			stRotationOptions.additionalTurns := 0;
			stRotationOptions.direction		  := Tc3_Mc3PlanarMotion.MC_Direction.mcDirectionNonModulo;

			IF NOT ipMoverApplication[nMoverIndex].std.P_MoveC.Busy THEN
					
				ipMoverApplication[nMoverIndex].std.MoveC( strInfo,
														   fRotationAngle,
														   fRotationVelocity,
														   fRotationAcceleration,
														   fRotationAcceleration,
														   fRotationJerk,
														   stRotationOptions );
														   
				nStateProcess := nStateProcess +1;
			END_IF										   

	211:	// Checking move command return
			IF ipMoverApplication[nMoverIndex].std.P_MoveC.Done THEN
				nStateProcess := nStateProcess +9;
			ELSIF ipMoverApplication[nMoverIndex].std.P_MoveC.Error THEN
				   nErrorID := ipMoverApplication[nMoverIndex].std.P_MoveOnTrack.ErrorID;
				  nObjectID := ipMoverApplication[nMoverIndex].std.P_MoveOnTrack.stInfo.nObjectID;
				nObjectType := ipMoverApplication[nMoverIndex].std.P_MoveOnTrack.stInfo.nObjectType;				
			END_IF			
			
				
	220:	// Process: Rotation-Demo done
			nStateProcess := 300;

		
			
			
	300: 	// Send mover to the next station
			fMoverToTrackPosition   := fSendAwayPosition;	
			nTrackIndex        		:= nStationTrackIndex;		
			fMoverVelocity     		:=    300.0;
			fMoverAcceleration 		:=  1_000.0;
			fMoverJerk         		:= 10_000.0;	
	
			
			stMoveParameters.direction := Tc3_Mc3PlanarMotion.MC_DIRECTION.mcDirectionPositive;	
			stMoveParameters.gap       := 240.0;

			
			// Creating info text with a little history of what happened in the station for debugging purpose		
			strInfo := fbHistoryInfo.CreateStationInfo(nStationIndex, nMoverIndex, nNextStationIndex);	
			
				
			// Move on track command	
			ipMoverApplication[nMoverIndex].std.MoveOnTrack( strInfo,
															 ipTrack[nTrackIndex].std,
															 fMoverToTrackPosition,
															 fMoverVelocity,
															 fMoverAcceleration,
															 fMoverJerk,
															 stMoveParameters.gap,
															 stMoveParameters.direction);
			nStateProcess := nStateProcess +1;
			
		
		
	301: 	// Checking move command return
			IF ipMoverApplication[nMoverIndex].std.P_MoveOnTrack.Active
			OR ipMoverApplication[nMoverIndex].std.P_MoveOnTrack.Done 
			THEN
				nStateProcess := nStateProcess + 9;
				
			ELSIF ipMoverApplication[nMoverIndex].std.P_MoveOnTrack.Error THEN
				   nErrorID := ipMoverApplication[nMoverIndex].std.P_MoveOnTrack.ErrorID;
				  nObjectID := ipMoverApplication[nMoverIndex].std.P_MoveOnTrack.stInfo.nObjectID;
				nObjectType := ipMoverApplication[nMoverIndex].std.P_MoveOnTrack.stInfo.nObjectType;
			END_IF		
		
			
	310: 	// Mover to the list of the next station
			ipStation[nNextStationIndex].P_List_Switch_Input_C.AddMover(P_List_Station.RemoveFirstInList());
			nStateProcess := 500;	
	
		
	500: 	// Done for this cycle
			nStateProcess := 100;

END_CASE
END_METHOD

END_FUNCTION_BLOCK

// ---- 2_Application/Station/FB_Station_03_Process.TcPOU
FUNCTION_BLOCK FB_Station_03_Process EXTENDS FB_StationBase
VAR
	nStationIndex				: UINT;
	nNextStationIndex			: UINT;
	nStationTrackIndex			: UINT;
	
	fStationPosition_X 			: LREAL;
	fStationPosition_Y 			: LREAL;		  
    fSendAwayDistance			: LREAL;	
	fInRangeDistance			: LREAL;	
	fSendAwayPosition			: LREAL;
	
	position					: PositionXYC;

END_VAR

METHOD Clear : BOOL
VAR_INPUT
END_VAR



	CASE nStateClear OF
		
	0:	// Enter
		Clear := FALSE;
		nStateClear := nStateClear +10;
		
	10: // Clearing all Station-Lists 
		IF SUPER^.Clear() THEN
			nStateClear := nStateClear +10;
		END_IF	
	
	20:	// Add aditional Data to be cleared here...
		nStateClear := 100;
		
		
	100: // Done
		      Clear := TRUE;
		nStateClear := 0;

	END_CASE
END_METHOD

METHOD Init : BOOL



VAR_INST
	nTestCounter	: INT;	
END_VAR
nTestCounter := nTestCounter +1;

CASE nStateInit OF

	0:		// Enter 
			bStationInitDone := FALSE;
			   nStateProcess := 0;
			      nStateInit := 10;
				 
			
	10:		// Init Station-Parameters				
				  nStationIndex := 3;				// Each station needs an unique index	
			 nStationTrackIndex := 3;	 			// Track on which the station resides
			  nNextStationIndex := 5;				// Index of the following station 
							  
			 fStationPosition_X := 840.0;			// Position of the station in X/Y coordinates
			 fStationPosition_Y := 360.0;			// Position of the station in X/Y coordinates
			  
			  fSendAwayDistance := 300.0;			// Position on track a mover will be send to after processing 
			  fInRangeDistance  := 300.0;			// Position in front of a station from where a mover will be taken over
			  
			  nStateInit := 11;
				   
				  
	11: // Fail-safe check, just to make sure all variables have been assigned after doing copy&paste from the template
			IF        nStationIndex > 0
			AND  nStationTrackIndex > 0
			AND   nNextStationIndex > 0
			AND  fStationPosition_X > 0
			AND  fStationPosition_Y > 0
			AND   fSendAwayDistance > 0
			THEN   
				nStateInit := 20;
			END_IF
			
				   
	20:		// Calculating positions
	
			// 1. Calculating station position on track
			position.SetValuesXYC(fStationPosition_X, fStationPosition_Y, 0.0);
			fStationPositionOnTrack := ipTrack[nStationTrackIndex].std.GetTrackPositionAt(position);
							
			// 2. Calculating send-away position on track
			fSendAwayPosition := fStationPositionOnTrack + fSendAwayDistance; 
			
			// The send away position must not exceed the lenght of the track!
			IF fSendAwayPosition > ipTrack[nStationTrackIndex].P_TrackLength THEN
				fSendAwayPosition := ipTrack[nStationTrackIndex].P_TrackLength;
			END_IF
			
			// 3. Calculating the station position in X/Y coordinates determined by the track	
            //    This is to make sure the center of the station is always located directly on the track.
			//    This value can differ from the initial fStationPosition_X, fStationPosition_Y in case they were not matching the track
			ipTrack[nStationTrackIndex].std.GetMoverPositionAt(fStationPositionOnTrack, StationPosition);
			
			// Providing the station position to e.g. visualization	
			stStationPosition.bInit            := TRUE;
			stStationPosition.fPositionOnTrack := fStationPositionOnTrack;
			stStationPosition.nTrackId         := nStationTrackIndex;
			stStationPosition.fPosition_X	   := StationPosition.x;
			stStationPosition.fPosition_Y	   := StationPosition.y;

			nStateInit := 30;
			
			
	30:		// Clear Lists
			IF THIS^.Clear() THEN
				nStateInit := 90;	
			END_IF

			
		
	90:		// Creating a little history of what happened in the station for debugging purpose
			fbHistoryInfo.AddEntry('Init');
	
			nStateInit := 100;
			
						
	100:	// Init done
			IF SUPER^.Init() THEN
				bStationInitDone := TRUE;	
				           Init := TRUE;
			END_IF
				
	
END_CASE
END_METHOD

METHOD Process : BOOL

VAR_INST
		
	nMoverIndex				: UINT;
	
	fMoverToTrackPosition	: LREAL;
	nTrackIndex				: UINT;
	fMoverVelocity			: LREAL;
	fMoverAcceleration		: LREAL;
	fMoverJerk				: LREAL;
	
	
	nErrorId					: UDINT;
	nObjectID					: UDINT;
	nObjectType					: UDINT;		
	
	// Process
	Timer01						: TON;
	fRotationAngle				: LREAL;
	fRotationVelocity			: LREAL;	
	fRotationAcceleration		: LREAL;
	fRotationJerk				: LREAL;
	stRotationOptions			: ST_MoveCOptions;
	
	fbRandom					: DRAND;
	fRandom						: LREAL;
	nRandom						: INT;
	
	bMoverGoodToGo				: BOOL;
	
	
	
END_VAR




VAR_INST



//	bToggleSwitch				: BOOL;
//	bStationActive				: BOOL;


//	fPositionOnTrack			: LREAL;
//	nCurrentTrackIndex			: UDINT;
	


//	fInRangePosition			: LREAL;
//	fOutOfRangePosition			: LREAL;
	


	
	
	
//	strInfo						: STRING;
	
					
	

//	ClearTrig					: R_TRIG;
	
//	TrackInfo					: PlanarObjectInfo;
//	nStationTrackID				: UDINT;
//	nMoverOnTrackID				: UDINT;
	

	
//	stMoveOptionsCurve			: ST_MoveCOptions;
//	fVeloTurn           		: LREAL :=   180.0;
//	fAccelTurn    				: LREAL :=  1000.0;
//	fJerkTurn            		: LREAL := 10000.0;	
//	fTurnAngle					: LREAL;	
	

END_VAR


// *** Processing Station ***

CASE nStateProcess OF 

	0:		// Enter
			IF bStationInitDone THEN
				nStateProcess := 100;
			END_IF

	
	100: 	// Waiting for Mover
			IF P_List_Station.P_FirstInList <> 0 THEN
				nMoverIndex := P_List_Station.P_FirstInList.P_Id;
					 nStateProcess := nStateProcess +10;
			END_IF
	
		
	110: 	// Check if Mover is in range
			IF  ipMoverApplication[nMoverIndex].std.P_SetOnTrack.TrackOID = ipTrack[nStationTrackIndex].std.P_OID 
			AND ipMoverApplication[nMoverIndex].std.P_SetOnTrack.SetPos   > fStationPositionOnTrack - fInRangeDistance
			THEN
				nStateProcess := nStateProcess +10;
			END_IF
			
	
	120: 	// Checking process situation
			CASE eProcessMode OF
				
			E_ProcessMode.None:
				;	// Nothing happens -> Process mode needs to be set!
				
			E_ProcessMode.InitRun:
				IF nStationIndex = 1 THEN
					ipMoverApplication[nMoverIndex].P_ProductData.bInitRun := FALSE;
				ELSE
					nStateProcess := 300;
				END_IF				
			
			E_ProcessMode.Production:
				nStateProcess := 200;
		
			END_CASE
		
	
	200: 	// Send mover to Processing-Position
			fMoverToTrackPosition   := fStationPositionOnTrack;
			nTrackIndex        		:= nStationTrackIndex;
			fMoverVelocity     		:=    300.0;
			fMoverAcceleration 		:=  1_000.0;
			fMoverJerk         		:= 10_000.0;	
	
			stMoveParameters.direction := Tc3_Mc3PlanarMotion.MC_DIRECTION.mcDirectionShortestWay;
			stMoveParameters.gap       := 200.0;
		
			
			// Creating info text with a little history of what happened in the station for debugging purpose		
			strInfo := fbHistoryInfo.CreateStationInfo(nStationIndex, nMoverIndex, nNextStationIndex);	


			// Move on track command	
			ipMoverApplication[nMoverIndex].std.MoveOnTrack( strInfo,
															 ipTrack[nTrackIndex].std,
															 fMoverToTrackPosition,
															 fMoverVelocity,
															 fMoverAcceleration,
															 fMoverJerk,
															 stMoveParameters.gap,
															 stMoveParameters.direction);
			nStateProcess := nStateProcess +1;
				
			
	201: 	// Checking move command return
			IF ipMoverApplication[nMoverIndex].std.P_MoveOnTrack.Done THEN
				nStateProcess := nStateProcess +9;
			ELSIF ipMoverApplication[nMoverIndex].std.P_MoveOnTrack.Error THEN
				   nErrorID := ipMoverApplication[nMoverIndex].std.P_MoveOnTrack.ErrorID;
				  nObjectID := ipMoverApplication[nMoverIndex].std.P_MoveOnTrack.stInfo.nObjectID;
				nObjectType := ipMoverApplication[nMoverIndex].std.P_MoveOnTrack.stInfo.nObjectType;
			END_IF		

			
	210:	// Process: Showing mover rotation -> Rotating 180°
			IF nRandom = 0 THEN
				fbRandom(seed := 0, Num=>fRandom);
				nRandom := LREAL_TO_INT(10*fRandom);
				nRandom := MAX(2,nRandom);
				IF nRandom > 8 THEN
					nRandom := -4;
				END_IF
			END_IF
			
			
			
			       fRotationAngle :=   90.0 * nRandom;
			    fRotationVelocity :=  360.0;
			fRotationAcceleration := 1800.0;
			        fRotationJerk := 9000.0;

			stRotationOptions.additionalTurns := 0;
			stRotationOptions.direction		  := Tc3_Mc3PlanarMotion.MC_Direction.mcDirectionNonModulo;

			IF NOT ipMoverApplication[nMoverIndex].std.P_MoveC.Busy THEN
					
				ipMoverApplication[nMoverIndex].std.MoveC( strInfo,
														   fRotationAngle,
														   fRotationVelocity,
														   fRotationAcceleration,
														   fRotationAcceleration,
														   fRotationJerk,
														   stRotationOptions );
				
			   	      nRandom := 0;										   
				nStateProcess := nStateProcess +1;
			END_IF										   

	211:	// Checking move command return
			IF ipMoverApplication[nMoverIndex].std.P_MoveC.Done THEN
				nStateProcess := nStateProcess +9;
			ELSIF ipMoverApplication[nMoverIndex].std.P_MoveC.Error THEN
				   nErrorID := ipMoverApplication[nMoverIndex].std.P_MoveOnTrack.ErrorID;
				  nObjectID := ipMoverApplication[nMoverIndex].std.P_MoveOnTrack.stInfo.nObjectID;
				nObjectType := ipMoverApplication[nMoverIndex].std.P_MoveOnTrack.stInfo.nObjectType;				
			END_IF			
			
				
	220:	// Process: Rotation-Demo done
			nStateProcess := 300;

				
	300:	// Check if the next station is ready to receive a mover
			IF eProcessMode = E_ProcessMode.Production THEN
				IF ipStation[nNextStationIndex].P_ProcessClearance = 0 THEN
					ipStation[nNextStationIndex].P_ProcessRequest := nStationIndex;
					nStateProcess := nStateProcess +1;	
				END_IF					
			ELSE
				nStateProcess := nStateProcess +10;
			END_IF
	
	301:	IF ipStation[nNextStationIndex].P_ProcessClearance = nStationIndex THEN
				nStateProcess := nStateProcess +9;	
			ELSIF ipStation[nNextStationIndex].P_ProcessRequest <> nStationIndex THEN
				nStateProcess := nStateProcess -1;
			END_IF
					
		
	310: 	// Send mover to the next station
			fMoverToTrackPosition   := fSendAwayPosition;	
			nTrackIndex        		:= nStationTrackIndex;		
			fMoverVelocity     		:=    300.0;
			fMoverAcceleration 		:=  1_000.0;
			fMoverJerk         		:= 10_000.0;	
	
			
			stMoveParameters.direction := Tc3_Mc3PlanarMotion.MC_DIRECTION.mcDirectionPositive;	
			stMoveParameters.gap       := 240.0;

			
			// Creating info text with a little history of what happened in the station for debugging purpose		
			strInfo := fbHistoryInfo.CreateStationInfo(nStationIndex, nMoverIndex, nNextStationIndex);	
			
				
			// Move on track command	
			ipMoverApplication[nMoverIndex].std.MoveOnTrack( strInfo,
															 ipTrack[nTrackIndex].std,
															 fMoverToTrackPosition,
															 fMoverVelocity,
															 fMoverAcceleration,
															 fMoverJerk,
															 stMoveParameters.gap,
															 stMoveParameters.direction);
			nStateProcess := nStateProcess +1;
			
		
		
	311: 	// Checking move command return
			IF ipMoverApplication[nMoverIndex].std.P_MoveOnTrack.Active
			OR ipMoverApplication[nMoverIndex].std.P_MoveOnTrack.Done 
			THEN
				nStateProcess := nStateProcess + 9;
				
			ELSIF ipMoverApplication[nMoverIndex].std.P_MoveOnTrack.Error THEN
				   nErrorID := ipMoverApplication[nMoverIndex].std.P_MoveOnTrack.ErrorID;
				  nObjectID := ipMoverApplication[nMoverIndex].std.P_MoveOnTrack.stInfo.nObjectID;
				nObjectType := ipMoverApplication[nMoverIndex].std.P_MoveOnTrack.stInfo.nObjectType;
			END_IF		
		
			
	320: 	// Mover to the list of the next station
			ipStation[nNextStationIndex].P_List_Switch_Input_B.AddMover(P_List_Station.RemoveFirstInList());
			nStateProcess := 500;	
	
		
	500: 	// Done for this cycle
			nStateProcess := 100;

END_CASE
END_METHOD

END_FUNCTION_BLOCK

// ---- 2_Application/Station/FB_Station_04_SW_Separate.TcPOU
FUNCTION_BLOCK FB_Station_04_SW_Separate EXTENDS FB_StationBase

VAR
	nStationIndex				: UINT;
	nPreviousStationIndexInputA : UINT;	
	nTrackIndexInputA 			: UINT;		
	nNextStationIndexOutputB 	: UINT;	
	nTrackIndexOutputB 			: UINT;		
	nNextStationIndexOutputC 	: UINT;	
	nTrackIndexOutputC 			: UINT;		
	
	fStationPosition_X 			: LREAL;
	fStationPosition_Y 			: LREAL;
	fInRangeDistance			: LREAL;		  
    fSendAwayDistanceOutputB    : LREAL;
	fSendAwayDistanceOutputC    : LREAL;	
	fSendAwayPositionOutputB	: LREAL;
	fSendAwayPositionOutputC	: LREAL;	

	position					: PositionXYC;

END_VAR

METHOD Clear : BOOL
VAR_INPUT
END_VAR



	CASE nStateClear OF
		
	0:	// Enter
		Clear := FALSE;
		nStateClear := nStateClear +10;
		
	10: // Clearing all Station-Lists 
		IF SUPER^.Clear() THEN
			nStateClear := nStateClear +10;
		END_IF	
	
	20:	// Add aditional Data to be cleared here...
		nStateClear := 100;
		
		
	100: // Done
		      Clear := TRUE;
		nStateClear := 0;

	END_CASE
END_METHOD

METHOD Init : BOOL



VAR_INST
	nTestCounter	: INT;	
END_VAR
nTestCounter := nTestCounter +1;

CASE nStateInit OF

	0:		// Enter 
			bStationInitDone := FALSE;
			   nStateProcess := 0;
			      nStateInit := 10;
				 
			
	10:		// Init Station-Parameters				
					       nStationIndex := 4;		// Each station needs an unique index		
			 nPreviousStationIndexInputA := 1;		// Index of the previous station on input_A		
				       nTrackIndexInputA := 1;		// Track on which the previous station resides	
			    nNextStationIndexOutputB := 3;		// Index of the following station on output_B		
				      nTrackIndexOutputB := 3;		// Track on which the following station resides
			    nNextStationIndexOutputC := 2;		// Index of the following station on output_C	
				      nTrackIndexOutputC := 2;		// Track on which the following station resides	 
			
                    fInRangeDistance := 300.0;		// Position in front of a station from where a mover will be taken over			  
		    fSendAwayDistanceOutputB := 300.0;		// Position on track a mover will be send to after processing 
		    fSendAwayDistanceOutputC := 300.0;		// Position on track a mover will be send to after processing 
		
			  nStateInit := 11;

			   
	11: // Fail-safe check, just to make sure all variables have been assigned after doing copy&paste from the template
			IF              nStationIndex > 0
			AND   nPreviousStationIndexInputA > 0	
			AND         nTrackIndexInputA > 0
			AND  nNextStationIndexOutputB > 0
			AND        nTrackIndexOutputB > 0
			AND  nNextStationIndexOutputC > 0
			AND        nTrackIndexOutputC > 0					
			AND          fInRangeDistance > 0
			AND  fSendAwayDistanceOutputB > 0
			AND  fSendAwayDistanceOutputC > 0
			THEN   
				nStateInit := 20;
			END_IF
			
				   
	20:		// Calculating positions
	
			// 1. Calculating station position on track
			fStationPositionOnTrack := ipTrack[nTrackIndexInputA].P_TrackLength;
							
			// 2. Calculating send-away position on track
			fSendAwayPositionOutputB := fSendAwayDistanceOutputB; 
			fSendAwayPositionOutputC := fSendAwayDistanceOutputC;
			
			// The send away position must not exceed the lenght of the following track!
			fSendAwayPositionOutputB := MIN(fSendAwayPositionOutputB, ipTrack[nTrackIndexOutputB].P_TrackLength);
			fSendAwayPositionOutputC := MIN(fSendAwayPositionOutputC, ipTrack[nTrackIndexOutputC].P_TrackLength);
			
					
			// 3. Calculating the station position in X/Y coordinates determined by the track	
            //    This is to make sure the center of the station is always located directly on the track.
			ipTrack[nTrackIndexInputA].std.GetMoverPositionAt(fStationPositionOnTrack, StationPosition);
			
			// Providing the station position to e.g. visualization	
			stStationPosition.bInit            := TRUE;
			stStationPosition.fPositionOnTrack := fStationPositionOnTrack;
			stStationPosition.nTrackId         := nTrackIndexOutputB;
			stStationPosition.fPosition_X	   := StationPosition.x;
			stStationPosition.fPosition_Y	   := StationPosition.y;

			nStateInit := 30;
			
			
	30:		// Clear Lists
			IF THIS^.Clear() THEN
				nStateInit := 90;	
			END_IF

			
		
	90:		// Creating a little history of what happened in the station for debugging purpose
			fbHistoryInfo.AddEntry('Init');
	
			nStateInit := 100;
			
						
	100:	// Init done
			IF SUPER^.Init() THEN
				bStationInitDone := TRUE;	
				           Init := TRUE;
			END_IF
				
	
END_CASE
END_METHOD

METHOD Process : BOOL

VAR_INST
		
	nMoverIndex				: UINT;
	
	fMoverToTrackPosition	: LREAL;
	nTrackIndex				: UINT;
	fMoverVelocity			: LREAL;
	fMoverAcceleration		: LREAL;
	fMoverJerk				: LREAL;
	
	
	nErrorId				: UDINT;
	nObjectID				: UDINT;
	nObjectType				: UDINT;		
	
	
	// Process
	nDestinationProcess		: UINT;
	nIncommingTrackOID		: UDINT;
	nNextStationIndex		: UINT;		 				
	fSendAwayPosition		: LREAL;
	nTrackindexNext			: UINT;
	
	
END_VAR

// Station - Switch-Seperate

CASE nStateProcess OF 

	0:		// Enter
			IF bStationInitDone THEN
				nStateProcess := 100;
			END_IF

	
	100: 	// Waiting for Mover
			IF P_List_Switch_Input_A.P_FirstInList <> 0 THEN
				P_List_Station.AddMover(P_List_Switch_Input_A.RemoveFirstInList());
			    nStateProcess := nStateProcess +10;
			END_IF
	
			
	110:	// Working with the station list from here on	
			IF P_List_Station.P_FirstInList <> 0 THEN
				nMoverIndex := P_List_Station.P_FirstInList.P_Id;
			    nStateProcess := nStateProcess +10;
			END_IF		
			
			
	120: 	// Check if Mover is in range
			IF  ipMoverApplication[nMoverIndex].std.P_SetOnTrack.TrackOID = ipTrack[nTrackIndexInputA].std.P_OID
			AND ipMoverApplication[nMoverIndex].std.P_SetOnTrack.SetPos   > fStationPositionOnTrack - fInRangeDistance
			THEN
				nStateProcess := nStateProcess +10;
			END_IF
			
			
			
	130: // Decide to which Station the mover has to travel to next.	
			nDestinationProcess := ipMoverApplication[nMoverIndex].P_ProductData.nDestinationProcess;	
			nIncommingTrackOID	:= ipMoverApplication[nMoverIndex].std.P_SetOnTrack.TrackOID;
			nTrackindex := 0;
						
			CASE nDestinationProcess OF
			0: // -> OutputB
				nNextStationIndex  := nNextStationIndexOutputB;
				fSendAwayPosition  := fSendAwayPositionOutputB;
				nTrackindexNext    := nTrackIndexOutputB;		
		
			2: // -> OutputC
				nNextStationIndex  := nNextStationIndexOutputC;
				fSendAwayPosition  := fSendAwayPositionOutputC;
				nTrackindexNext    := nTrackIndexOutputC;				
	
			3: // -> OutputB
				nNextStationIndex  := nNextStationIndexOutputB;
				fSendAwayPosition  := fSendAwayPositionOutputB;
				nTrackindexNext    := nTrackIndexOutputB;		
			END_CASE
			
			IF nTrackindexNext > 0 THEN
				nStateProcess := 200;	
			END_IF
			
			
		
	200: 	// Send mover to the next station	
			fMoverToTrackPosition := fSendAwayPosition;
			nTrackIndex           := nTrackindexNext;
			fMoverVelocity     	  :=    300.0;
			fMoverAcceleration 	  :=  1_000.0;
			fMoverJerk         	  := 10_000.0;	
	
			stMoveParameters.direction := Tc3_Mc3PlanarMotion.MC_DIRECTION.mcDirectionPositive;	
			stMoveParameters.gap       := 240.0;

			
			// Creating info text with a little history of what happened in the station for debugging purpose		
			strInfo := fbHistoryInfo.CreateStationInfo(nStationIndex, nMoverIndex, nNextStationIndex);	
			
				
			// Move on track command	
			ipMoverApplication[nMoverIndex].std.MoveOnTrack( strInfo,
															 ipTrack[nTrackIndex].std,
															 fMoverToTrackPosition,
															 fMoverVelocity,
															 fMoverAcceleration,
															 fMoverJerk,
															 stMoveParameters.gap,
															 stMoveParameters.direction);
			nStateProcess := nStateProcess +1;
			
		
		
	201: 	// Checking move command return
			IF ipMoverApplication[nMoverIndex].std.P_MoveOnTrack.Active
			OR ipMoverApplication[nMoverIndex].std.P_MoveOnTrack.Done 
			THEN
				nStateProcess := nStateProcess + 9;
				
			ELSIF ipMoverApplication[nMoverIndex].std.P_MoveOnTrack.Error THEN
				   nErrorID := ipMoverApplication[nMoverIndex].std.P_MoveOnTrack.ErrorID;
				  nObjectID := ipMoverApplication[nMoverIndex].std.P_MoveOnTrack.stInfo.nObjectID;
				nObjectType := ipMoverApplication[nMoverIndex].std.P_MoveOnTrack.stInfo.nObjectType;
			END_IF		
		
	
	210:	// Wait till the mover passed the junction point
			IF ipMoverApplication[nMoverIndex].std.P_SetOnTrack.TrackOID <> ipTrack[nTrackIndexInputA].std.P_OID THEN
				nStateProcess := nStateProcess + 10;
			END_IF		

		
	220: 	// Mover to the list of the next station
			ipStation[nNextStationIndex].P_List_Station.AddMover(P_List_Station.RemoveFirstInList());
			nStateProcess := 500;	
	
		
	500: 	// Done for this cycle
			nStateProcess := 100;

END_CASE
END_METHOD

END_FUNCTION_BLOCK

// ---- 2_Application/Station/FB_Station_05_SW_Merge.TcPOU
FUNCTION_BLOCK FB_Station_05_SW_Merge EXTENDS FB_StationBase
VAR
	nStationIndex				: UINT;
	nNextStationIndexOutputA 	: UINT;	
	nNextStationIndex			: UINT;
	nTrackIndexOutputA 			: UINT;		
	
	fStationPosition_X 			: LREAL;
	fStationPosition_Y 			: LREAL;		  
    fSendAwayDistance			: LREAL;	
	fInRangeDistance			: LREAL;	
	fSendAwayPosition			: LREAL;
	
	position					: PositionXYC;

END_VAR

METHOD Clear : BOOL
VAR_INPUT
END_VAR



	CASE nStateClear OF
		
	0:	// Enter
		Clear := FALSE;
		nStateClear := nStateClear +10;
		
	10: // Clearing all Station-Lists 
		IF SUPER^.Clear() THEN
			nStateClear := nStateClear +10;
		END_IF	
	
	20:	// Add aditional Data to be cleared here...
		nStateClear := 100;
		
		
	100: // Done
		      Clear := TRUE;
		nStateClear := 0;

	END_CASE
END_METHOD

METHOD Init : BOOL



VAR_INST
	nTestCounter	: INT;	
END_VAR
nTestCounter := nTestCounter +1;

CASE nStateInit OF

	0:		// Enter 
			bStationInitDone := FALSE;
			   nStateProcess := 0;
			      nStateInit := 10;
				 
			
	10:		// Init Station-Parameters				
					   nStationIndex := 5;			// Each station needs an unique index				
			nNextStationIndexOutputA := 1;			// Index of the following station on output_A		
				  nTrackIndexOutputA := 1;			// Track on which the following station resides
				  		  
			      fStationPosition_X := 480.0;		// Position of the station in X/Y coordinates
			      fStationPosition_Y := 120.0;		// Position of the station in X/Y coordinates
			  
			       fSendAwayDistance := 300.0;		// Position on track a mover will be send to after processing 
			       fInRangeDistance  := 300.0;		// Position in front of a station from where a mover will be taken over
			  
			       nStateInit := 11;
  
			   
	11: // Fail-safe check, just to make sure all variables have been assigned after doing copy&paste from the template
			IF              nStationIndex > 0
			AND  nNextStationIndexOutputA > 0
			AND        nTrackIndexOutputA > 0				
			AND        fStationPosition_X > 0
			AND        fStationPosition_Y > 0
			AND         fSendAwayDistance > 0
			THEN   
				nStateInit := 20;
			END_IF
			
				   
	20:		// Calculating positions
	
			// 1. Calculating station position on track
			fStationPositionOnTrack := 0.0;
							
			// 2. Calculating send-away position on track
			fSendAwayPosition := fSendAwayDistance; 
			
			// The send away position must not exceed the lenght of the track!
			IF fSendAwayPosition > ipTrack[nTrackIndexOutputA].P_TrackLength THEN
				fSendAwayPosition := ipTrack[nTrackIndexOutputA].P_TrackLength;
			END_IF
			
			// 3. Calculating the station position in X/Y coordinates determined by the track	
            //    This is to make sure the center of the station is always located directly on the track.
			ipTrack[nTrackIndexOutputA].std.GetMoverPositionAt(fStationPositionOnTrack, StationPosition);
			
			// Providing the station position to e.g. visualization	
			stStationPosition.bInit            := TRUE;
			stStationPosition.fPositionOnTrack := fStationPositionOnTrack;
			stStationPosition.nTrackId         := nTrackIndexOutputA;
			stStationPosition.fPosition_X	   := StationPosition.x;
			stStationPosition.fPosition_Y	   := StationPosition.y;

			nStateInit := 30;
			
			
	30:		// Clear Lists
			IF THIS^.Clear() THEN
				nStateInit := 90;	
			END_IF

			
		
	90:		// Creating a little history of what happened in the station for debugging purpose
			fbHistoryInfo.AddEntry('Init');
	
			nStateInit := 100;
			
						
	100:	// Init done
			IF SUPER^.Init() THEN
				bStationInitDone := TRUE;	
				           Init := TRUE;
			END_IF
				
	
END_CASE
END_METHOD

METHOD Process : BOOL

VAR_INST
		
	nMoverIndex				: UINT;
	
	fMoverToTrackPosition	: LREAL;
	nTrackIndex				: UINT;
	fMoverVelocity			: LREAL;
	fMoverAcceleration		: LREAL;
	fMoverJerk				: LREAL;
	
	
	nErrorId				: UDINT;
	nObjectID				: UDINT;
	nObjectType				: UDINT;		
	
	
	// Process
	nMoverIndexInputB			: UINT;
	nMoverIndexInputC			: UINT;	
	
	bNewMoverIn					: BOOL;
	
	
	(*
	nDestinationProcess		: UINT;
	nIncommingTrackOID		: UDINT;
	nNextStationIndex		: UINT;		 				
	fSendAwayPosition		: LREAL;
	nTrackindexNext			: UINT;
	*)
	
	
END_VAR

// Station - Switch-Merge

CASE nStateProcess OF 

	0:		// Enter
			IF bStationInitDone THEN
				nStateProcess := 100;
			END_IF

						
	100:	// Clearance
			IF eProcessMode = E_ProcessMode.Production THEN
				nProcessClearence := 0;
				IF nProcessRequest > 0 THEN
					nProcessClearence := nProcessRequest;
					  nProcessRequest := 0;
						nStateProcess := nStateProcess +5;
				ELSE
					IF P_List_Switch_Input_B.P_FirstInList <> 0	
					OR P_List_Switch_Input_C.P_FirstInList <> 0
					THEN
						nStateProcess := nStateProcess +5;	
					END_IF
				END_IF
			ELSE
				nStateProcess := nStateProcess +5;	
			END_IF

		
	105: 	// Waiting for Mover on Input_B or Input_C
	            nProcessState := 0;
			      nMoverIndex := 0;
			nMoverIndexInputB := 0;
			nMoverIndexInputC := 0;
			      bNewMoverIn := FALSE;
	
			IF P_List_Switch_Input_B.P_FirstInList <> 0 THEN
				nMoverIndexInputB := P_List_Switch_Input_B.P_FirstInList.P_Id;
			END_IF		
			
			IF P_List_Switch_Input_C.P_FirstInList <> 0 THEN
				nMoverIndexInputC := P_List_Switch_Input_C.P_FirstInList.P_Id;
			END_IF		
		
			// Copy mover data to station list, Input_B is prioritized
			IF nMoverIndexInputB > 0 THEN
				P_List_Station.AddMover(P_List_Switch_Input_B.RemoveFirstInList());
				bNewMoverIn := TRUE;
			ELSIF nMoverIndexInputC > 0 THEN
				P_List_Station.AddMover(P_List_Switch_Input_C.RemoveFirstInList());
				bNewMoverIn := TRUE;
			END_IF
			
			IF bNewMoverIn THEN
				nProcessState := 1;
				nStateProcess := nStateProcess +5;
			END_IF
			
			
	110:	// Working with the station list from here on:
			nMoverIndex := 0;
			IF P_List_Station.P_FirstInList <> 0 THEN
				nMoverIndex := P_List_Station.P_FirstInList.P_Id;
			END_IF
						
			IF nMoverIndex > 0 THEN
				nNextStationIndex := nNextStationIndexOutputA;
				    nStateProcess := nStateProcess +10;
			END_IF
			
			
	120: 	// Check if Mover is in range
			IF ipMoverApplication[nMoverIndex].std.P_SetOnTrack.SetPos > fStationPositionOnTrack - fInRangeDistance THEN
				nStateProcess := 200;
			END_IF
			

			
		
	200: 	// Send mover to the next station	
			fMoverToTrackPosition := fSendAwayPosition;
			nTrackIndex           := nTrackIndexOutputA;
			fMoverVelocity     	  :=    300.0;
			fMoverAcceleration 	  :=  1_000.0;
			fMoverJerk         	  := 10_000.0;	
	
			stMoveParameters.direction := Tc3_Mc3PlanarMotion.MC_DIRECTION.mcDirectionPositive;	
			stMoveParameters.gap       := 240.0;

			
			// Creating info text with a little history of what happened in the station for debugging purpose		
			strInfo := fbHistoryInfo.CreateStationInfo(nStationIndex, nMoverIndex, nNextStationIndex);	
			
				
			// Move on track command	
			ipMoverApplication[nMoverIndex].std.MoveOnTrack( strInfo,
															 ipTrack[nTrackIndex].std,
															 fMoverToTrackPosition,
															 fMoverVelocity,
															 fMoverAcceleration,
															 fMoverJerk,
															 stMoveParameters.gap,
															 stMoveParameters.direction);
			nStateProcess := nStateProcess +1;
			
		
		
	201: 	// Checking move command return
			IF ipMoverApplication[nMoverIndex].std.P_MoveOnTrack.Active
			OR ipMoverApplication[nMoverIndex].std.P_MoveOnTrack.Done 
			THEN
				nStateProcess := nStateProcess + 9;
				
			ELSIF ipMoverApplication[nMoverIndex].std.P_MoveOnTrack.Error THEN
				   nErrorID := ipMoverApplication[nMoverIndex].std.P_MoveOnTrack.ErrorID;
				  nObjectID := ipMoverApplication[nMoverIndex].std.P_MoveOnTrack.stInfo.nObjectID;
				nObjectType := ipMoverApplication[nMoverIndex].std.P_MoveOnTrack.stInfo.nObjectType;
			END_IF		
		
			
	210:	// Wait till the mover passed the junction point
			IF ipMoverApplication[nMoverIndex].std.P_SetOnTrack.TrackOID = ipTrack[nTrackIndexOutputA].std.P_OID THEN
				nStateProcess := nStateProcess + 10;
			END_IF		
			
			
	220: 	// Mover to the list of the next station
			ipStation[nNextStationIndex].P_List_Station.AddMover(P_List_Station.RemoveFirstInList());
			nStateProcess := 500;	
	
		
	500: 	// Done for this cycle
			nStateProcess := 100;

END_CASE
END_METHOD

END_FUNCTION_BLOCK

// ---- 1_Industry/FB_SK_StateManager.TcPOU
FUNCTION_BLOCK FB_SK_StateManager

VAR
	bStartUpDone		: BOOL;	
	bFirstAbortDone		: BOOL;
	
	eCommand			: E_XMotion_Command;	
	eCommandOld			: E_XMotion_Command;
	eStatus				: E_XMotion_Status;	
	nCommandCounter		: UDINT;

END_VAR

METHOD PUBLIC Cycle
VAR_INPUT
END_VAR


	IF NOT bStartUpDone THEN					
		eStatus := E_XMotion_Status.StartUp;
	ELSIF NOT bFirstAbortDone THEN
		eStatus := E_XMotion_Status.Aborting;
	ELSE

		IF eCommand <> eCommandOld THEN
			eCommandOld := eCommand;
	
			nCommandCounter := nCommandCounter +1;
			
			
			CASE eCommand OF
				
			
			E_XMotion_Command.Abort:	
						eStatus := E_XMotion_Status.Aborting;	
			
			E_XMotion_Command.Reset:
						IF eStatus = E_XMotion_Status.Aborted THEN
							eStatus := E_XMotion_Status.Resetting;	
						END_IF
				
			E_XMotion_Command.Prepare:
						IF eStatus = E_XMotion_Status.Stopped THEN
							eStatus := E_XMotion_Status.Preparing;	
						END_IF	
			
			E_XMotion_Command.Start:
						IF eStatus = E_XMotion_Status.Prepared THEN
							eStatus := E_XMotion_Status.Execute;	
						END_IF	

			E_XMotion_Command.HoldOnError:
						eStatus := E_XMotion_Status.HoldOnError;

					
			END_CASE
		END_IF
		
	END_IF
END_METHOD

METHOD PUBLIC StateComplete : BOOL
VAR_INPUT
END_VAR




	CASE eStatus OF
		
	E_XMotion_Status.StartUp:
				bStartUpDone := TRUE;
				
	E_XMotion_Status.Aborting:
				bFirstAbortDone := TRUE;	
				eStatus := E_XMotion_Status.Aborted;	
	
	E_XMotion_Status.Resetting:
				eStatus := E_XMotion_Status.Stopped;
		
	E_XMotion_Status.Preparing:
				eStatus := E_XMotion_Status.Prepared;
	
				
	END_CASE
END_METHOD

PROPERTY Status : E_XMotion_Status
GET
Status := eStatus;
END_GET
END_PROPERTY

PROPERTY XMotionCommand : E_XMotion_Command
SET
eCommand := XMotionCommand;
END_SET
END_PROPERTY

END_FUNCTION_BLOCK

// ---- 1_Industry/FB_OperationalControl.TcPOU
FUNCTION_BLOCK FB_OperationalControl
VAR_INPUT

	bStartCommand 		: BOOL;
	bStopCommand 		: BOOL;		
	bQuitCommand 		: BOOL;
	bExceptionCommand	: BOOL;
	bResetCommand		: BOOL;

END_VAR
VAR_OUTPUT
	bStartLamp 			: BOOL;
	bStopLamp 			: BOOL;
	bQuitLamp 			: BOOL;
	bEStopLamp			: BOOL;
	bStopping			: BOOL;
	bStopped			: BOOL;
	bStarting 			: BOOL;
	bRunning			: BOOL;
	sResult 			: STRING;
	nResult				: INT;
END_VAR

VAR_IN_OUT
	XTags		: ST_XTags;
END_VAR

VAR
	nMachineState		: INT;
	bStartUpFlag		: BOOL;
	bStartUpDone		: BOOL;
	bError				: BOOL;
	bStartSequence		: BOOL;
	bStopSequence		: BOOL;
	bStartLampBlink		: BOOL;
	bStopLampBlink		: BOOL;
	nErrorSequence		: INT;
	tBlinker			: TON;
	bBlinker			: BOOL;

	bCheckCurrentMachineState	: BOOL;

	nProcessFeedback		: UDINT;

	rtMoverErrordetection	: R_TRIG;
	bMoverErrorDetected		: BOOL;
	
	rtReset					: R_TRIG;
	bDoReset				: BOOL;
	
END_VAR


	helper();

	rtReset(CLK:=bResetCommand);
	IF rtReset.Q THEN
		IF bMoverErrorDetected THEN
			bDoReset := TRUE;
		END_IF
	END_IF
	

	// Check for system start-up
	IF NOT bStartUpDone THEN
		IF XTags.Status = E_XMotion_Status.StartUp THEN
			bStartUpFlag := TRUE;
		END_IF			
		IF bStartUpFlag AND XTags.Status = E_XMotion_Status.Aborted THEN	
			IF NOT bStartUpDone THEN
				bStartUpDone   := TRUE;
			    bStartSequence := FALSE;
		        bStopSequence  := TRUE;
			END_IF
		END_IF	
		sResult := 'Machine Start-Up';
	END_IF
	

	// Check start signal
	IF bStartCommand 
	AND NOT bStopCommand 
	AND NOT bExceptionCommand
	AND NOT bStopSequence
	AND NOT bError
	THEN 
		bStartSequence := TRUE;
		bStopSequence  := FALSE;
	END_IF
	
	// Check stop signal
	IF bStopCommand 
	AND NOT bExceptionCommand
	AND NOT bError
	THEN
		bStartSequence := FALSE;
		bStopSequence  := TRUE;
	END_IF 
	
		
	ErrorSequence();
	StartSequence();
	StopSequence();
	SyncSequence();

ACTION ErrorSequence:
	
CASE nErrorSequence OF
		
	0:	// Checking mover error  
		IF ipMotionSystemApplication <> 0 THEN
			rtMoverErrordetection(CLK:=ipMotionSystemApplication.P_MoverError);
			IF rtMoverErrordetection.Q THEN
				bMoverErrorDetected := TRUE;
			END_IF
		END_IF	
		
		// In case of an exception e.g. E-Stop, start the error sequence
		IF bExceptionCommand THEN    // -> Exception from extern e.g. E-Stop Button
			XTags.Command := E_XMotion_Command.Abort;
			nErrorSequence := 5;
		ELSE
			IF bMoverErrorDetected THEN	// -> Exception from a Mover e.g. FollowingError
				XTags.Command := E_XMotion_Command.HoldOnError;
				nErrorSequence := 5;
			END_IF			
		END_IF	

		
	5:	// In case of an exception e.g. E-Stop, start the error sequence
		 bStartSequence := FALSE;
		 bStopSequence  := FALSE;
			 bStartLamp := FALSE;
			  bStopLamp := FALSE;
			  bQuitLamp := FALSE;
		bStartLampBlink := FALSE;
		 bStopLampBlink := FALSE;	 
				 bError := TRUE;	
		
	     nErrorSequence := 10;
		
	
	10:	// Waiting till the event is gone e.g. E-Stop has been pulled out.		
		bEStopLamp := bBlinker;
		sResult := 'Error pending';	
		IF NOT bExceptionCommand THEN
			    bEStopLamp := FALSE;
			nErrorSequence := 20;
		END_IF
			
		
	20:	// Wait for error-quit	
		bQuitLamp := bBlinker;
		
		IF ipMotionSystemApplication.P_MoverError THEN
			sResult := 'Mover Error / Waiting for error-quit';
		ELSE
			sResult := 'Waiting for error-quit';
		END_IF

		IF bExceptionCommand THEN
			nErrorSequence := 5;
		ELSIF bQuitCommand THEN
			bMoverErrorDetected := FALSE;
			     nErrorSequence := 30;
		ELSIF bDoReset THEN
			           bDoReset := FALSE;
			bMoverErrorDetected := FALSE;
			     nErrorSequence := 40;			
		END_IF
		
		
	30: // Sending abort-command to the StarterKit-StateMachine.
		XTags.Command := E_XMotion_Command.Abort;
		     bQuitLamp := bBlinker;
		       sResult := 'Error-Quit - sending abort-command';		
		nErrorSequence := 40;
		
	  
	40: // Waiting for StarterKit-StateMachine in state Aborted.
		IF XTags.Status = E_XMotion_Status.Aborted THEN
			bQuitLamp := FALSE;
		    bStopLamp := TRUE;
			   bError := FALSE;
			  sResult := 'Error-Quit successful';	
			  
			nErrorSequence := 0;
		END_IF		  

	END_CASE
END_ACTION

ACTION helper:




	IF bStartLampBlink THEN
		bStartLamp := bBlinker;
	END_IF
	
	IF bStopLampBlink THEN
		bStopLamp := bBlinker;
	END_IF
	

	tBlinker(IN:=TRUE, PT:=T#500MS);
	IF tBlinker.Q THEN
		bBlinker := NOT bBlinker;
		tBlinker(IN:=FALSE);
	END_IF
END_ACTION

PROPERTY P_ProcessFeedback : UDINT
SET
nProcessFeedback := P_ProcessFeedback;
END_SET
END_PROPERTY

ACTION StartSequence:


	
	
	
	// Start-Sequence, will run in case of start-signal 
	IF bStartSequence THEN
		CASE XTags.Status OF
			
			E_XMotion_Status.StartUp:	// Do nothing
										bStartSequence := FALSE;
										sResult := 'Impossible - Machine is still in Start-Up procedure';	
										
			E_XMotion_Status.Aborting:	// Do nothing
										bStartSequence := FALSE;
										sResult := 'Impossible - Machine is in Aborting sequence';	
		
			E_XMotion_Status.Aborted:	// Reset-Command brings you to the next stage
										  nMachineState := 1;
										bStartLampBlink := TRUE;
										      bStopLamp := FALSE;
										  XTags.Command := E_XMotion_Command.Reset;
										sResult := 'Starting - command reset issued';
		
			E_XMotion_Status.Resetting: // Wait for next stage
			  						      nMachineState := 1;
										bStartLampBlink := TRUE;
										      bStopLamp := FALSE;
										sResult := 'Starting - Machine is resetting';
										
			E_XMotion_Status.Stopped:	// Prepare-Command brings you to the next stage
									      nMachineState := 2;
										bStartLampBlink := TRUE;
										  XTags.Command := E_XMotion_Command.Prepare;
										sResult := 'Starting - command prepare issued';	
		
			E_XMotion_Status.Preparing: // Wait for next stage
										  nMachineState := 3;
										bStartLampBlink := TRUE;
										      bStopLamp := FALSE;
										sResult := 'Starting - Machine is preparing';
		
			E_XMotion_Status.Prepared:	// Start-Command brings you to the next stage
										  nMachineState := 3;
										bStartLampBlink := TRUE;
										      bStopLamp := FALSE;
										  XTags.Command := E_XMotion_Command.Start;
										sResult := 'Starting - command start issued';	 
		
			E_XMotion_Status.Execute:	// System is running
										 nMachineState := 4;
									   bStartLampBlink := FALSE;
											 bStopLamp := FALSE;
										    bStartLamp := TRUE;
										bStartSequence := FALSE;
										sResult := 'Machine is running';
		
		END_CASE
	END_IF
END_ACTION

ACTION StopSequence:





	

	// Stop-Sequence, will run in case of stop-signal 
	IF bStopSequence THEN
		     bStartLamp := FALSE;
		bStartLampBlink := FALSE;
		
		CASE XTags.Status OF
			
			E_XMotion_Status.StartUp:	// Do nothing
										bStopSequence := FALSE;
										sResult := 'Impossible - Machine is still in Start-Up procedure';	
										
			E_XMotion_Status.Aborting:	// Do nothing
										sResult := 'Impossible - Machine is in Aborting sequence';	
		
			E_XMotion_Status.Aborted:	// System is stopped
										 nMachineState := 2;
			                            bStopLampBlink := FALSE;
			                                 bStopLamp := TRUE;
										 bStopSequence := FALSE;
										sResult := 'Machine is stopped';
		
			E_XMotion_Status.Resetting: // Sending abort-command
										 nMachineState := 1;
										bStopLampBlink := TRUE;
										 XTags.Command := E_XMotion_Command.Abort;
										sResult := 'Machine is resetting - sending abort-command';
										
			E_XMotion_Status.Stopped:	// Sending abort-command
										 nMachineState := 1;
										bStopLampBlink := TRUE;
										 XTags.Command := E_XMotion_Command.Abort;
										sResult := 'Machine is stopped - sending abort-command';
		
			E_XMotion_Status.Preparing: // Sending abort-command
										 nMachineState := 1;
										 nMachineState := 1;
										bStopLampBlink := TRUE;
										 XTags.Command := E_XMotion_Command.Abort;
										sResult := 'Machine is preparing - sending abort-command';
		
			E_XMotion_Status.Prepared:	// Sending abort-command
										 nMachineState := 1;
										bStopLampBlink := TRUE;
										 XTags.Command := E_XMotion_Command.Abort;
										sResult := 'Machine is prepared - sending abort-command';
		
			E_XMotion_Status.Execute:	// Sending abort-command
									     nMachineState := 1;
										bStopLampBlink := TRUE;
										    bStartLamp := FALSE;
										 XTags.Command := E_XMotion_Command.Abort;
										sResult := 'Machine is executing - sending abort-command';
		
		END_CASE

	END_IF
END_ACTION

ACTION SyncSequence:




	

	CASE nMachineState OF
		
	0:	// Machine state = undefined
		bStopping := FALSE;
		bStopped  := FALSE;
		bStarting := FALSE;
		bRunning  := FALSE;	
				
	1:	// Machine state = stopping	
		bStopping := TRUE;
		bStopped  := FALSE;
		bStarting := FALSE;
		bRunning  := FALSE;	
		IF XTags.Status <> E_XMotion_Status.Aborting THEN
			bCheckCurrentMachineState := TRUE;
		END_IF
		
	2:	// Machine state = stopped	
		bStopping := FALSE;
		bStopped  := TRUE;
		bStarting := FALSE;
		bRunning  := FALSE;	
		IF XTags.Status <> E_XMotion_Status.Stopped THEN
			bCheckCurrentMachineState := TRUE;
		END_IF
	
	3:	// Machine state = starting	
		bStopping := FALSE;
		bStopped  := FALSE;
		bStarting := TRUE;
		bRunning  := FALSE;
		IF XTags.Status <> E_XMotion_Status.Preparing THEN
			bCheckCurrentMachineState := TRUE;
		END_IF					
		
	4:	// Machine state = running	
		bStopping := FALSE;
		bStopped  := FALSE;
		bStarting := FALSE;
		bRunning  := TRUE;		
		IF XTags.Status <> E_XMotion_Status.Execute THEN
			bCheckCurrentMachineState := TRUE;
		END_IF
		
	END_CASE



	// Syncronizing with StarterKit-StateMachine
	IF bCheckCurrentMachineState 
	AND NOT bError
	THEN
		bCheckCurrentMachineState := FALSE;
		
		CASE XTags.Status OF
			
			E_XMotion_Status.StartUp:	// Do nothing
										sResult := 'Machine Start-Up';
										
										bStartSequence := FALSE;
										 bStopSequence := FALSE;
										 nMachineState := 0;
											
										
			E_XMotion_Status.Aborting:	// Do nothing
										        sResult := 'Machine Aborting';	
										  nMachineState := 1;
										bStartLampBlink := FALSE;
										     bStartLamp := FALSE;
										 bStopLampBlink := TRUE;
										      bStopLamp := FALSE;
		
			E_XMotion_Status.Aborted:	// Reset-Command brings you to the next stage
										        sResult := 'Machine Aborted';	
										  nMachineState := 2;
										bStartLampBlink := FALSE;
										     bStartLamp := FALSE;
										 bStopLampBlink := FALSE;
										      bStopLamp := TRUE;

		
			E_XMotion_Status.Resetting: // Wait for next stage
										        sResult := 'Machine Resetting';	
			  						      nMachineState := 1;
										bStartLampBlink := TRUE;
										      bStopLamp := FALSE;

										
			E_XMotion_Status.Stopped:	// Prepare-Command brings you to the next stage
									   	        sResult := 'Stopped';
									      nMachineState := 2;
	
		
			E_XMotion_Status.Preparing: // Wait for next stage
												sResult := 'Machine Preparing';
										  nMachineState := 3;
										bStartLampBlink := TRUE;
										      bStopLamp := FALSE;

		
			E_XMotion_Status.Prepared:	// Start-Command brings you to the next stage
										        sResult := 'Prepared';
										  nMachineState := 3;
										bStartLampBlink := TRUE;
										      bStopLamp := FALSE;
	 
		
			E_XMotion_Status.Execute:	// System is running
									           sResult := 'Machine is Running';
										 nMachineState := 4;
									   bStartLampBlink := FALSE;
											 bStopLamp := FALSE;
										    bStartLamp := TRUE;
										bStartSequence := FALSE;
		
		END_CASE
	END_IF
END_ACTION

END_FUNCTION_BLOCK

// ---- 1_Industry/FB_VisStarterKitStateMachine.TcPOU
FUNCTION_BLOCK FB_VisStarterKitStateMachine

VAR_IN_OUT

	iq_stVisControl  : ST_VisControl;
	iq_XTags		 : ST_XTags;
		
END_VAR





VAR
		
	diStatusOld : DINT := -1;
	
	
	// Operator-Control-Pad 
	bOCStartButton			: BOOL;
	bOCStopButton			: BOOL;
	bOCQuitButton			: BOOL;
	bOCEStopButton			: BOOL;
	
	bOCStopLamp				: BOOL;
	bOCStartLamp			: BOOL;
	bOCQuitLamp				: BOOL;
	bOCEStopLamp			: BOOL;
	
	bOCMessageColorGreen	: BOOL;
	bOCMessageColorRed		: BOOL;	
	
	sOCResultText			: STRING;
	sDisplayText			: STRING;
	nStringPosition			: INT;
	nStringLength			: INT;
	nDisplayLenght			: INT := 28;
		
	nOCResultNumber			: INT;
	DisplayTimer			: TON;
	
	rtNoCommandTrigger		: R_TRIG;
	
	bInitScreenDone			: BOOL;
	nVisArrangement			: INT;
	nVisArrangementMem		: INT;
	nVisArrangementSet		: INT;
	
END_VAR




	ScreenArrangement();
	
	StarterKitStateMachine();

	OperatorInterface();

ACTION OperatorInterface:



	

		
		
		bOCStartButton 	:= iq_stVisControl.stOperatorPad.bStartButtunState;
		bOCStopButton  	:= iq_stVisControl.stOperatorPad.bStopButtonState; 
		bOCQuitButton	:= iq_stVisControl.stOperatorPad.bQuitButtonState;
		bOCEStopButton	:= iq_stVisControl.stOperatorPad.bEStopButtonState;
		
		
		iq_stVisControl.stOperatorPad.bStartButtonLamp 		:= bOCStartLamp;
		iq_stVisControl.stOperatorPad.bStopButtonLamp  		:= bOCStopLamp;
		iq_stVisControl.stOperatorPad.bQuitButtonLamp  		:= bOCQuitLamp;
		iq_stVisControl.stOperatorPad.bEStopButtonLamp 		:= bOCEStopLamp;
		iq_stVisControl.stOperatorPad.bMessageColorGreen 	:= bOCMessageColorGreen;
		iq_stVisControl.stOperatorPad.bMessageColorRed   	:= bOCMessageColorRed;
		
			
		nStringLength := LEN(sOCResultText);	
		IF nStringLength > nDisplayLenght THEN
			sDisplayText := MID(sOCResultText,nDisplayLenght,nStringPosition);
		
			DisplayTimer(IN:=TRUE, PT:=T#500MS);
			IF DisplayTimer.Q THEN
				DisplayTimer(IN:=FALSE);
				nStringPosition := nStringPosition +1;
				
				IF nStringPosition > (nStringLength - nDisplayLenght) THEN
					nStringPosition := 1;
				END_IF
			END_IF
		ELSE
			sDisplayText := sOCResultText;
		END_IF
		iq_stVisControl.stOperatorPad.sMessage := sDisplayText;
END_ACTION

PROPERTY PUBLIC P_OCEStopButtonState : BOOL
GET
P_OCEStopButtonState := bOCEStopButton;
END_GET
END_PROPERTY

PROPERTY PUBLIC P_OCEStopLampState : BOOL
SET
bOCEStopLamp := P_OCEStopLampState;
END_SET
END_PROPERTY

PROPERTY PUBLIC P_OCQuitButtonState : BOOL
GET
P_OCQuitButtonState := bOCQuitButton;
END_GET
END_PROPERTY

PROPERTY PUBLIC P_OCQuitLampState : BOOL
SET
bOCQuitLamp := P_OCQuitLampState;
END_SET
END_PROPERTY

PROPERTY PUBLIC P_OCResult : int
SET
nOCResultNumber := P_OCResult;
END_SET
END_PROPERTY

PROPERTY PUBLIC P_OCResultTextDisplay : STRING
SET
sOCResultText := P_OCResultTextDisplay;
END_SET
END_PROPERTY

PROPERTY PUBLIC P_OCStartButtonState : BOOL
GET
P_OCStartButtonState := bOCStartButton;
END_GET
END_PROPERTY

PROPERTY PUBLIC P_OCStartLampState : BOOL
SET
bOCStartLamp := P_OCStartLampState;
END_SET
END_PROPERTY

PROPERTY PUBLIC P_OCStopButtonState : BOOL
GET
P_OCStopButtonState := bOCStopButton;
END_GET
END_PROPERTY

PROPERTY PUBLIC P_OCStopLampState : BOOL
SET
bOCStopLamp := P_OCStopLampState;
END_SET
END_PROPERTY

ACTION ScreenArrangement:






	// Decide which Pad shall be shown at system boot:
	IF NOT bInitScreenDone THEN
		bInitScreenDone := TRUE;

		iq_stVisControl.stControlPad.bVisInvisibleButton  := FALSE;		
		iq_stVisControl.stOperatorPad.bVisInvisibleButton := FALSE;
	END_IF


	// Check which Pad shall be shown right now:
	IF iq_stVisControl.stControlPad.bVisInvisibleButton THEN
		iq_stVisControl.stControlPad.bVisInvisible := TRUE;
	ELSE
		iq_stVisControl.stControlPad.bVisInvisible := FALSE;
	END_IF	

	IF iq_stVisControl.stOperatorPad.bVisInvisibleButton THEN
		iq_stVisControl.stOperatorPad.bVisInvisible := TRUE;
	ELSE
		iq_stVisControl.stOperatorPad.bVisInvisible := FALSE;
	END_IF		
	

	// Determine current visualisation arrangement:
	IF  iq_stVisControl.stControlPad.bVisInvisible 
	AND iq_stVisControl.stOperatorPad.bVisInvisible
	THEN
		nVisArrangement := 1;
		
	ELSIF ( NOT iq_stVisControl.stControlPad.bVisInvisible
			AND iq_stVisControl.stOperatorPad.bVisInvisible) 
	THEN
		nVisArrangement := 2;
		
	ELSIF ( NOT iq_stVisControl.stOperatorPad.bVisInvisible 
			AND iq_stVisControl.stControlPad.bVisInvisible )
	THEN
		nVisArrangement := 3;
	ELSIF (     NOT iq_stVisControl.stControlPad.bVisInvisible 
			AND NOT iq_stVisControl.stOperatorPad.bVisInvisible)
	THEN
		nVisArrangement := 4;
	END_IF
	
	
	
	// Arranging all frame positions according to current arrangement:
	IF nVisArrangement <> nVisArrangementMem THEN
		nVisArrangementMem := nVisArrangement;
		nVisArrangementSet := nVisArrangement;
	END_IF
		
	CASE nVisArrangementSet OF 	
	
	1:  nVisArrangementSet := 0;
		
		iq_stVisControl.stControlPad.nFramePositionX   :=  0;
		iq_stVisControl.stControlPad.nFramePositionY   :=  0;
		iq_stVisControl.stControlPad.nButtonPositionX  :=  0;
		iq_stVisControl.stControlPad.nButtonPositionY  := 55;
		
		iq_stVisControl.stOperatorPad.nFramePositionX  :=  0;
		iq_stVisControl.stOperatorPad.nFramePositionY  :=  0;
		iq_stVisControl.stOperatorPad.nButtonPositionX :=  0;
		iq_stVisControl.stOperatorPad.nButtonPositionY := 55;
				
	2: 	nVisArrangementSet := 0;
	
		iq_stVisControl.stControlPad.nFramePositionX   :=  0;
		iq_stVisControl.stControlPad.nFramePositionY   := 60;	
		iq_stVisControl.stOperatorPad.nButtonPositionX :=  0;
		iq_stVisControl.stOperatorPad.nButtonPositionY := 55;	
	
	3:	nVisArrangementSet := 0;
	
		iq_stVisControl.stControlPad.nButtonPositionX  :=  0;
		iq_stVisControl.stControlPad.nButtonPositionY  := -2;
		iq_stVisControl.stOperatorPad.nFramePositionX  :=  0;
		iq_stVisControl.stOperatorPad.nFramePositionY  :=  0;
	
	4:	nVisArrangementSet := 0;
	
		iq_stVisControl.stControlPad.nFramePositionX   :=  0;
		iq_stVisControl.stControlPad.nFramePositionY   :=  0;
		iq_stVisControl.stOperatorPad.nFramePositionX  :=  0;
		iq_stVisControl.stOperatorPad.nFramePositionY  :=  0;
	
	END_CASE
END_ACTION

ACTION StarterKitStateMachine:


	// Setting XTag-Commands according to user-commands
	IF    iq_stVisControl.stControlPad.bButtonState_Abort THEN
				rtNoCommandTrigger(CLK:=FALSE);
				iq_XTags.Command  := E_XMotion_Command.Abort;	
	ELSIF iq_stVisControl.stControlPad.bButtonState_Reset THEN
				rtNoCommandTrigger(CLK:=FALSE);
				iq_XTags.Command  := E_XMotion_Command.Reset;	
	ELSIF iq_stVisControl.stControlPad.bButtonState_Prepare THEN
				rtNoCommandTrigger(CLK:=FALSE);
				iq_XTags.Command  := E_XMotion_Command.Prepare;	
	ELSIF iq_stVisControl.stControlPad.bButtonState_Start THEN
				rtNoCommandTrigger(CLK:=FALSE);
				iq_XTags.Command  := E_XMotion_Command.Start;	
	ELSE
			rtNoCommandTrigger(CLK:=TRUE);
			IF rtNoCommandTrigger.Q THEN
				iq_XTags.Command  := E_XMotion_Command.NoCommand;
			END_IF
	END_IF


	
	
	// Setting Vis display according to current status	
	iq_stVisControl.stControlPad.iAbortSequenceState   := iq_XTags.States.nAbortState;
	iq_stVisControl.stControlPad.iResetSequenceState   := iq_XTags.States.nResetState;
	iq_stVisControl.stControlPad.iPrepareSequenceState := iq_XTags.States.nPrepareState;
	iq_stVisControl.stControlPad.iStartSequenceState   := iq_XTags.States.nStartState;
	

	IF iq_XTags.Status <> diStatusOld THEN
		diStatusOld := iq_XTags.Status;	
	
		iq_stVisControl.stControlPad.bAbortSequenceStateInvisible 	:= TRUE;
		iq_stVisControl.stControlPad.bResetSequenceStateInvisible 	:= TRUE;
		iq_stVisControl.stControlPad.bPrepareSequenceStateInvisible := TRUE;
		iq_stVisControl.stControlPad.bStartSequenceStateInvisible	:= TRUE;
		
		iq_stVisControl.stControlPad.bStateSignalAbortBlue     := FALSE;
		iq_stVisControl.stControlPad.bStateSignalAbortYellow   := FALSE;
		iq_stVisControl.stControlPad.bStateSignalAbortGreen    := FALSE;
		iq_stVisControl.stControlPad.bStateSignalResetYellow   := FALSE;
		iq_stVisControl.stControlPad.bStateSignalResetGreen    := FALSE;		
		iq_stVisControl.stControlPad.bStateSignalResetYellow   := FALSE;
		iq_stVisControl.stControlPad.bStateSignalResetGreen    := FALSE;		
		iq_stVisControl.stControlPad.bStateSignalPrepareYellow := FALSE;
		iq_stVisControl.stControlPad.bStateSignalPrepareGreen  := FALSE;		
		iq_stVisControl.stControlPad.bStateSignalExecuteYellow := FALSE;
		iq_stVisControl.stControlPad.bStateSignalExecuteGreen  := FALSE;	

		IF 	   iq_XTags.Status = E_XMotion_Status.Aborting THEN
					iq_stVisControl.stControlPad.bAbortSequenceStateInvisible := FALSE;
					iq_stVisControl.stControlPad.bStateSignalAbortYellow   	  := TRUE;		
		ELSIF iq_XTags.Status = E_XMotion_Status.Aborted THEN
					iq_stVisControl.stControlPad.bStateSignalAbortGreen := TRUE;
		ELSIF iq_XTags.Status = E_XMotion_Status.Resetting THEN
					iq_stVisControl.stControlPad.bResetSequenceStateInvisible := FALSE;
					iq_stVisControl.stControlPad.bStateSignalResetYellow      := TRUE;
		ELSIF iq_XTags.Status = E_XMotion_Status.Stopped THEN
					iq_stVisControl.stControlPad.bStateSignalResetGreen := TRUE;
		ELSIF iq_XTags.Status = E_XMotion_Status.Preparing THEN
					iq_stVisControl.stControlPad.bPrepareSequenceStateInvisible := FALSE;
					iq_stVisControl.stControlPad.bStateSignalPrepareYellow      := TRUE;
		ELSIF iq_XTags.Status = E_XMotion_Status.Prepared THEN
					iq_stVisControl.stControlPad.bStateSignalPrepareGreen := TRUE;
		ELSIF iq_XTags.Status = E_XMotion_Status.Execute THEN
					iq_stVisControl.stControlPad.bStartSequenceStateInvisible := FALSE;
					iq_stVisControl.stControlPad.bStateSignalExecuteGreen     := TRUE;
		ELSIF iq_XTags.Status = E_XMotion_Status.StartUp THEN
					iq_stVisControl.stControlPad.bStateSignalAbortBlue := TRUE;
		END_IF	

	END_IF
END_ACTION

END_FUNCTION_BLOCK

// ---- 1_Industry/VISUs/OperationalControlPad.TcVIS
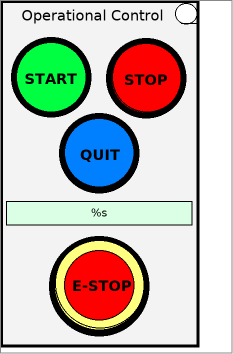
VISUALIZATION OperationalControlPad  // 233x354
VAR_IN_OUT
	stVisOperationalControl	: ST_Vis_OperationalControl;
END_VAR
    Rectangle (0,0 199x347)
    Label (9,1 167x29), "Operational Control"
    Ellipse (11,37 80x80)
    Ellipse (16,42 70x70)
    Ellipse (16,42 70x70), invisible if: NOT stVisOperationalControl.bStartButtonLamp
    Ellipse (106,38 80x80)
    Ellipse (111,43 70x70)
    Ellipse (111,43 70x70), invisible if: Not stVisOperationalControl.bStopButtonLamp
    Ellipse (59,113 80x80)
    Ellipse (64,118 70x70)
    Ellipse (64,118 70x70), invisible if: NOT stVisOperationalControl.bQuitButtonLamp
    Label (13,64 76x30), "START"
    Label (108,65 76x30), "STOP"
    Label (62,140 76x30), "QUIT"
    Rectangle (6,201 186x24), "%s", text variable: stVisOperationalControl.sMessage
    Ellipse (49,236 100x100)
    Ellipse (54,240 90x90)
    Ellipse (64,250 70x70)
    Ellipse (64,250 70x70), invisible if: NOT stVisOperationalControl.bEStopButtonLamp
    Label (64,271 76x30), "E-STOP"
    Rectangle (6,201 186x24), "%s", text variable: stVisOperationalControl.sMessage, invisible if: NOT stVisOperationalControl.bMessageColorRed
    Rectangle (6,201 186x24), "%s", text variable: stVisOperationalControl.sMessage, invisible if: NOT stVisOperationalControl.bMessageColorGreen
    Ellipse (16,42 70x70)
        tap stVisOperationalControl.bStartButtunState
    Ellipse (112,42 70x70)
        tap stVisOperationalControl.bStopButtonState
    Ellipse (64,117 70x70)
        tap stVisOperationalControl.bQuitButtonState
    Ellipse (55,238 90x90)
        toggle stVisOperationalControl.bEStopButtonState
    Ellipse (175,3 22x21)
    Line (218,-7) (233,-6)
    Line (181,23) (197,23)
    Rectangle (158,2 40x30)
        OnMouseClick: execute { stVisOperationalControl.bVisInvisibleButton := TRUE; }
END_VISUALIZATION

// ---- 1_Industry/VISUs/StarterKitStateMachinelPad.TcVIS
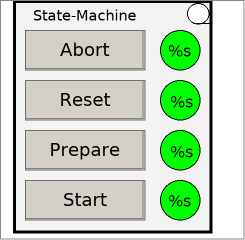
VISUALIZATION StarterKitStateMachinelPad  // 245x240
VAR_IN_OUT
	
	stControlPadControl		:   ST_Vis_ControlPadControl;

END_VAR
    Rectangle (13,0 199x233)
    Button (25,30 120x40), "Abort"
        tap stControlPadControl.bButtonState_Abort p3779583253=TRUE
    Button (25,80 120x40), "Reset"
        tap stControlPadControl.bButtonState_Reset
    Button (25,130 120x40), "Prepare"
        tap stControlPadControl.bButtonState_Prepare
    Button (25,180 120x40), "Start"
        tap stControlPadControl.bButtonState_Start
    Ellipse (160,30 40x40)
    Ellipse (160,30 40x40), invisible if: NOT stControlPadControl.bStateSignalAbortYellow
    Group (160,80 40x40)
        Ellipse (0,0 40x40)
        Ellipse (0,0 40x40), invisible if: NOT stControlPadControl.bStateSignalResetYellow
        Ellipse (0,0 40x40), invisible if: NOT stControlPadControl.bStateSignalResetGreen
    Group (160,130 40x40)
        Ellipse (0,0 40x40)
        Ellipse (0,0 40x40), invisible if: NOT stControlPadControl.bStateSignalPrepareYellow
        Ellipse (0,0 40x40), invisible if: NOT stControlPadControl.bStateSignalPrepareGreen
    Group (160,180 40x40)
        Ellipse (0,0 40x40)
        Ellipse (0,0 40x40), invisible if: NOT stControlPadControl.bStateSignalExecuteYellow
        Ellipse (0,0 40x40), invisible if: NOT stControlPadControl.bStateSignalExecuteGreen
    Ellipse (160,30 40x40), invisible if: NOT stControlPadControl.bStateSignalAbortBlue
    Ellipse (160,30 40x40), invisible if: NOT stControlPadControl.bStateSignalAbortGreen
    Label (19,1 132x29), "State-Machine"
    Textfield (159,35 42x32), "%s", text variable: stControlPadControl.iAbortSequenceState, invisible if: stControlPadControl.bAbortSequenceStateInvisible
    Textfield (161,86 42x32), "%s", text variable: stControlPadControl.iResetSequenceState, invisible if: stControlPadControl.bResetSequenceStateInvisible
    Textfield (161,136 42x32), "%s", text variable: stControlPadControl.iPrepareSequenceState, invisible if: stControlPadControl.bPrepareSequenceStateInvisible
    Textfield (159,185 42x32), "%s", text variable: stControlPadControl.iStartSequenceState, invisible if: stControlPadControl.bStartSequenceStateInvisible
    Ellipse (187,3 22x21)
    Line (230,-7) (245,-6)
    Line (193,23) (209,23)
    Rectangle (179,3 32x25)
        OnMouseClick: execute { stControlPadControl.bVisInvisibleButton := TRUE; }
END_VISUALIZATION

// ---- GlobalTextList.TcGTLO
TEXTLIST GlobalTextList
  632 = '\txPlanar'
  135 = '\tXPlanar'
  427 = '\nGroup\nNotReady'
  425 = '\nGroup\nStandby'
  140 = '%.3f'
  243 = '%d'
  602 = '%d /'
  145 = '%d Axes'
  43 = '%s'
  245 = '+'
  246 = '-'
  532 = '/'
  81 = '1'
  902 = '2'
  489 = '3'
  115 = '4'
  268 = '5'
  274 = 'A'
  39 = 'Abort'
  56 = 'Activated'
  726 = 'Activating'
  774 = 'ActivationState'
  215 = 'B'
  306 = 'Busy'
  671 = 'C'
  224 = 'CA_Group'
  560 = 'E-STOP'
  144 = 'Enable Requested FALSE'
  143 = 'Enable Requested TRUE'
  51 = 'Entrance Location'
  790 = 'Error in the Group or in one of the axes'
  789 = 'error on the\ngroup or in one\nof the axes'
  331 = 'Error: %d'
  1811 = 'Exit Location'
  146 = 'General'
  431 = 'Group\nErrorDisabled'
  430 = 'Group\nErrorEnabled'
  429 = 'GroupDisabled'
  428 = 'GroupErrorStop'
  424 = 'GroupMoving'
  426 = 'GroupStopping'
  750 = 'GVL_StationVisu.aMoverInQueue[INDEX]'
  748 = 'GVL_StationVisu.aMoverInSequence[INDEX].nMover'
  749 = 'GVL_StationVisu.aMoverInSequence[INDEX].nSequence'
  413 = 'GVL_XPlanarVisuDiag.aMoverInSequence[INDEX].nMover'
  498 = 'GVL_XPlanarVisuDiag.aMoverInSequence[INDEX].nSequence'
  53 = 'Home'
  152 = 'Inactive'
  142 = 'INVALID'
  938 = 'M1'
  303 = 'M2'
  38 = 'M3'
  609 = 'M4'
  432 = 'MC_AddAxis'
  783 = 'MC_GroupDisable'
  786 = 'MC_GroupEnable'
  784 = 'MC_GroupHalt'
  434 = 'MC_GroupReset'
  785 = 'MC_GroupStop'
  433 = 'MC_RemAxis'
  787 = 'MC_UngroupAllAxes'
  114 = 'Mover'
  348 = 'Mover:'
  522 = 'MoverId:'
  1100 = 'NumMoversReq.'
  788 = 'one axis\nnot ready'
  807 = 'OnTrack'
  105 = 'Operational Control'
  49 = 'Operational Control Pad'
  819 = 'PosA'
  255 = 'PosB'
  653 = 'PosC'
  207 = 'Position Check Failed! '
  217 = 'Position Check Failed!     Mover 3 too far away from rotation point.'
  372 = 'Position Check Failed! Mover 3 too far away from rotation point'
  837 = 'PosX'
  932 = 'PosY'
  30 = 'PosZ'
  953 = 'Prepare'
  927 = 'Process'
  1737 = 'Prozess Location'
  1111 = 'Queue'
  872 = 'Queue Location'
  509 = 'QueueGap'
  675 = 'QueuePositions'
  134 = 'QUIT'
  40 = 'Reset'
  42 = 'Run'
  407 = 'Show Rotation'
  41 = 'Start'
  678 = 'START'
  260 = 'State'
  390 = 'State-Machine'
  839 = 'State-Machine Pad'
  291 = 'Station'
  197 = 'Station Parameter'
  461 = 'Station: %d'
  1657 = 'Station: %s'
  141 = 'Status'
  939 = 'STOP'
  499 = 'Track'
  466 = 'Utility'
  791 = 'V 2.1'
  241 = 'V 3.0'
  233 = 'V 3.1'
  679 = 'V 3.2'
  970 = 'V 3.3'
  900 = 'X'
  984 = 'XPlanar Example Project'
  313 = 'y'
END_TEXTLIST

// ---- VISU/ControlXplanar/VI_Control_Xplanar.TcVIS
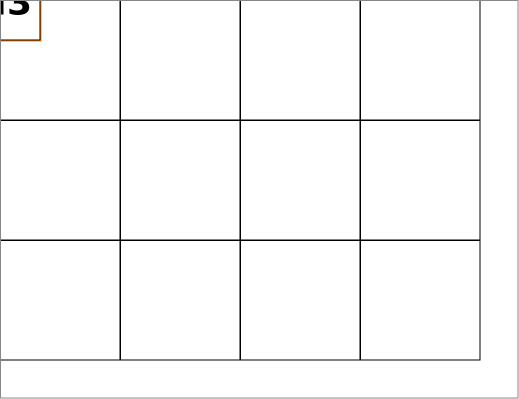
VISUALIZATION VI_Control_Xplanar  // 519x399
    Rectangle (0,0 120x120)
    Rectangle (120,0 120x120)
    Rectangle (240,0 120x120)
    Rectangle (360,0 120x120)
    Rectangle (0,120 120x120)
    Rectangle (120,120 120x120)
    Rectangle (240,120 120x120)
    Rectangle (360,120 120x120)
    Rectangle (0,240 120x120)
    Rectangle (120,240 120x120)
    Rectangle (240,240 120x120)
    Rectangle (360,240 120x120)
    Rectangle (-39,-39 80x80), "1", invisible if: NOT g_VisStationData[1].bInit
        p3560616238: g_VisStationData[1].fPosition_X/2
        p2738717112: (720-g_VisStationData[1].fPosition_Y)/2
    Rectangle (-39,-39 80x80), "2", invisible if: NOT g_VisStationData[2].bInit
        p3560616238: g_VisStationData[2].fPosition_X/2
        p2738717112: (720-g_VisStationData[2].fPosition_Y)/2
    Rectangle (-39,-39 80x80), "3", invisible if: NOT g_VisStationData[3].bInit
        p3560616238: g_VisStationData[3].fPosition_X/2
        p2738717112: (720-g_VisStationData[3].fPosition_Y)/2
    Rectangle (-39,-39 80x80), "4", invisible if: NOT g_VisStationData[4].bInit
        p3560616238: g_VisStationData[4].fPosition_X/2
        p2738717112: (720-g_VisStationData[4].fPosition_Y)/2
    Rectangle (-39,-39 80x80), "5", invisible if: NOT g_VisStationData[5].bInit
        p3560616238: g_VisStationData[5].fPosition_X/2
        p2738717112: (720-g_VisStationData[5].fPosition_Y)/2
    Rectangle (-37,-37 77x77), "M1"
        p3560616238: MAIN.fbXMotionUnit.fbMover[1].VisuPos.x/2
        p2738717112: (720-MAIN.fbXMotionUnit.fbMover[1].VisuPos.y)/2
        p2858320360: -MAIN.fbXMotionUnit.fbMover[1].VisuPos.c
    Rectangle (-37,-37 77x77), "M2"
        p3560616238: MAIN.fbXMotionUnit.fbMover[2].VisuPos.x/2
        p2738717112: (720-MAIN.fbXMotionUnit.fbMover[2].VisuPos.y)/2
        p2858320360: -MAIN.fbXMotionUnit.fbMover[2].VisuPos.c
    Rectangle (-37,-37 77x77), "M4"
        p3560616238: MAIN.fbXMotionUnit.fbMover[4].VisuPos.x/2
        p2738717112: (720-MAIN.fbXMotionUnit.fbMover[4].VisuPos.y)/2
        p2858320360: -MAIN.fbXMotionUnit.fbMover[4].VisuPos.c
    Rectangle (-37,-37 77x77), "M3"
        p3560616238: MAIN.fbXMotionUnit.fbMover[3].VisuPos.x/2
        p2738717112: (720-MAIN.fbXMotionUnit.fbMover[3].VisuPos.y)/2
        p2858320360: -MAIN.fbXMotionUnit.fbMover[3].VisuPos.c
END_VISUALIZATION

// ---- VISU/Pages/MessageBox_2.TcVIS
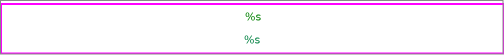
VISUALIZATION MessageBox_2  // 504x55
VAR_IN_OUT
	message_1 : ST_MessageBoxText;
	message_2 : ST_MessageBoxText;
END_VAR
    Textfield (3,2 500x30), "%s", text variable: message_1.sText
        p55702900: message_1.nColor
    Textfield (2,25 500x30), "%s", text variable: message_2.sText
        p55702900: message_2.nColor
    Rectangle (0,3 504x51)
        p3450524324: message_1.nColor
END_VISUALIZATION

// ---- VISU/Pages/MessageBox_1.TcVIS
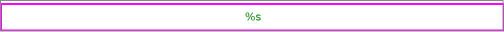
VISUALIZATION MessageBox_1  // 504x32
VAR_IN_OUT
	message_1 : ST_MessageBoxText;
END_VAR
    Textfield (3,2 500x30), "%s", text variable: message_1.sText
        p55702900: message_1.nColor
    Rectangle (0,3 504x28)
        p3450524324: message_1.nColor
END_VISUALIZATION

// ---- VISU/Pages/UtilityPage.TcVIS
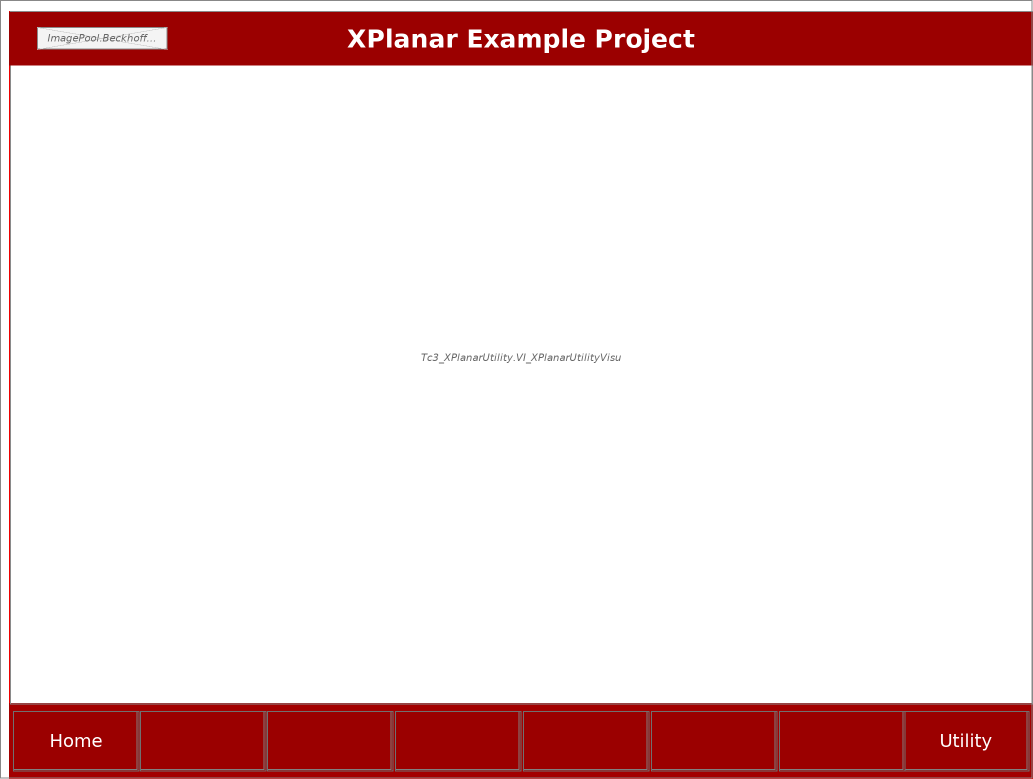
VISUALIZATION UtilityPage  // 1033x779
    Rectangle (9,11 1024x768)
    Rectangle (9,703 1024x75)
    Button (13,711 126x60), "Home"
        OnMouseDown: change screen: Visualization
    Button (140,711 126x60)
    Button (903,711 126x60), "Utility"
        OnMouseUp: change screen: UtilityPage
    Button (395,711 126x60)
    Button (523,711 126x60)
    Button (651,711 126x60)
    Button (779,711 126x60)
    Button (267,711 126x60)
    Frame (10,11 1023x693)
        shows Tc3_XPlanarUtility.VI_XPlanarUtilityVisu()
    Group (9,12 1024x53)
        Image (18,11 130x22), image: ImagePool.Beckhoff_white
        Rectangle (0,0 1024x53), "XPlanar Example Project"
        Image (28,15 130x22), image: ImagePool.Beckhoff_white
END_VISUALIZATION

// ---- VISU/Pages/VI_MainSide.TcVIS
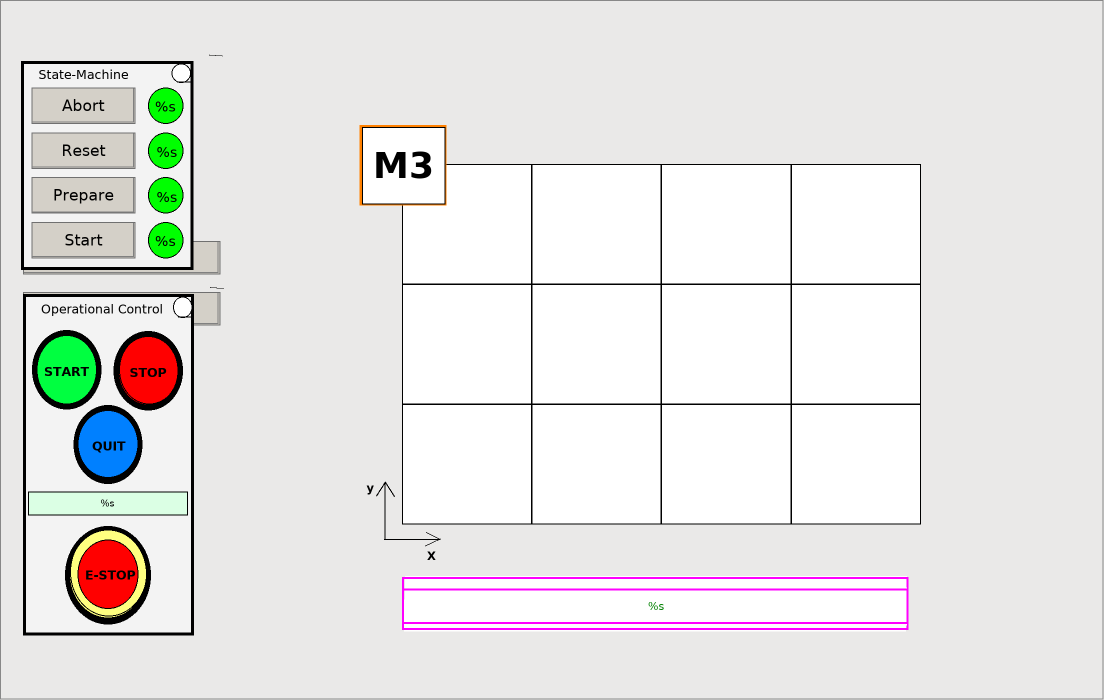
VISUALIZATION VI_MainSide  // 1104x700
    Polygon (172,381) (173,382)
    Frame (402,164 561x399)
        shows VI_Control_Xplanar()
    Button (23,292 197x33), "Operational Control Pad", invisible if: NOT stVisControl.stOperatorPad.bVisInvisible
        p3560616238: stVisControl.stOperatorPad.nButtonPositionX
        p2738717112: stVisControl.stOperatorPad.nButtonPositionY
        OnMouseClick: execute { stVisControl.stOperatorPad.bVisInvisibleButton := FALSE; }
    Button (23,241 197x33), "State-Machine Pad", invisible if: NOT stVisControl.stControlPad.bVisInvisible
        p3560616238: stVisControl.stControlPad.nButtonPositionX
        p2738717112: stVisControl.stControlPad.nButtonPositionY
        OnMouseClick: execute { stVisControl.stControlPad.bVisInvisibleButton := FALSE; }
    Frame (10,61 212x215), invisible if: stVisControl.stControlPad.bVisInvisible
        shows StarterKitStateMachinelPad(stControlPadControl := stVisControl.stControlPad)
        p3560616238: stVisControl.stControlPad.nFramePositionX
        p2738717112: stVisControl.stControlPad.nFramePositionY
    Frame (23,294 200x348), invisible if: stVisControl.stOperatorPad.bVisInvisible
        shows OperationalControlPad(stVisOperationalControl := stVisControl.stOperatorPad)
        p3560616238: stVisControl.stOperatorPad.nFramePositionX
        p2738717112: stVisControl.stOperatorPad.nFramePositionY
    Rectangle (1025,637 79x63)
    Group (357,473 88x98)
        Label (61,68 27x30), "X"
        Label (0,0 27x30), "y"
        Group (19,9 64x64)
            Line (8,57) (64,57)
            Line (50,50) (64,57)
            Line (64,57) (49,64)
            Line (9,57) (9,1)
            Line (9,0) (18,14)
            Line (9,0) (0,14)
    Frame (402,574 506x57), invisible if: NOT g_VisuMessage.bVisible_Box1_B
        shows MessageBox_2(message_1 := g_VisuMessage.sMessage_L1_Box1, message_2 := g_VisuMessage.sMessage_L2_Box1)
        tap g_VisuMessage.bAcknowledge
    Frame (402,585 506x40), invisible if: NOT g_VisuMessage.bVisible_Box1_A
        shows MessageBox_1(message_1 := g_VisuMessage.sMessage_L1_Box1)
END_VISUALIZATION

// ---- VISU/Pages/VI_MainSide_1.TcVIS
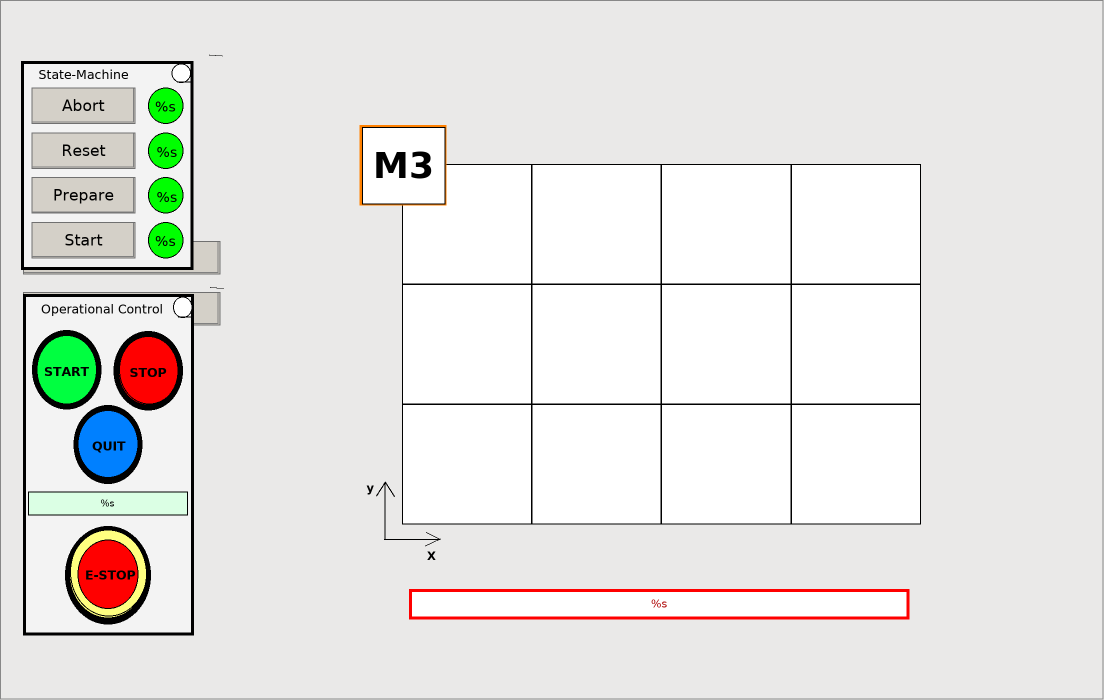
VISUALIZATION VI_MainSide_1  // 1104x700
    Polygon (172,381) (173,382)
    Frame (402,164 561x399)
        shows VI_Control_Xplanar()
    Button (23,292 197x33), "Operational Control Pad", invisible if: NOT stVisControl.stOperatorPad.bVisInvisible
        p3560616238: stVisControl.stOperatorPad.nButtonPositionX
        p2738717112: stVisControl.stOperatorPad.nButtonPositionY
        OnMouseClick: execute { stVisControl.stOperatorPad.bVisInvisibleButton := FALSE; }
    Button (23,241 197x33), "State-Machine Pad", invisible if: NOT stVisControl.stControlPad.bVisInvisible
        p3560616238: stVisControl.stControlPad.nButtonPositionX
        p2738717112: stVisControl.stControlPad.nButtonPositionY
        OnMouseClick: execute { stVisControl.stControlPad.bVisInvisibleButton := FALSE; }
    Frame (10,61 212x215), invisible if: stVisControl.stControlPad.bVisInvisible
        shows StarterKitStateMachinelPad(stControlPadControl := stVisControl.stControlPad)
        p3560616238: stVisControl.stControlPad.nFramePositionX
        p2738717112: stVisControl.stControlPad.nFramePositionY
    Frame (23,294 200x348), invisible if: stVisControl.stOperatorPad.bVisInvisible
        shows OperationalControlPad(stVisOperationalControl := stVisControl.stOperatorPad)
        p3560616238: stVisControl.stOperatorPad.nFramePositionX
        p2738717112: stVisControl.stOperatorPad.nFramePositionY
    Rectangle (1025,637 79x63)
    Group (357,473 88x98)
        Label (61,68 27x30), "X"
        Label (0,0 27x30), "y"
        Group (19,9 64x64)
            Line (8,57) (64,57)
            Line (50,50) (64,57)
            Line (64,57) (49,64)
            Line (9,57) (9,1)
            Line (9,0) (18,14)
            Line (9,0) (0,14)
    Textfield (409,589 500x30), "%s", text variable: MAIN.stVisAlarm.sAlarmMessage, invisible if: NOT MAIN.stVisAlarm.bAlarmActive
END_VISUALIZATION

// ---- VISU/Pages/VI_Tc3_XPlanarUtility.TcVIS
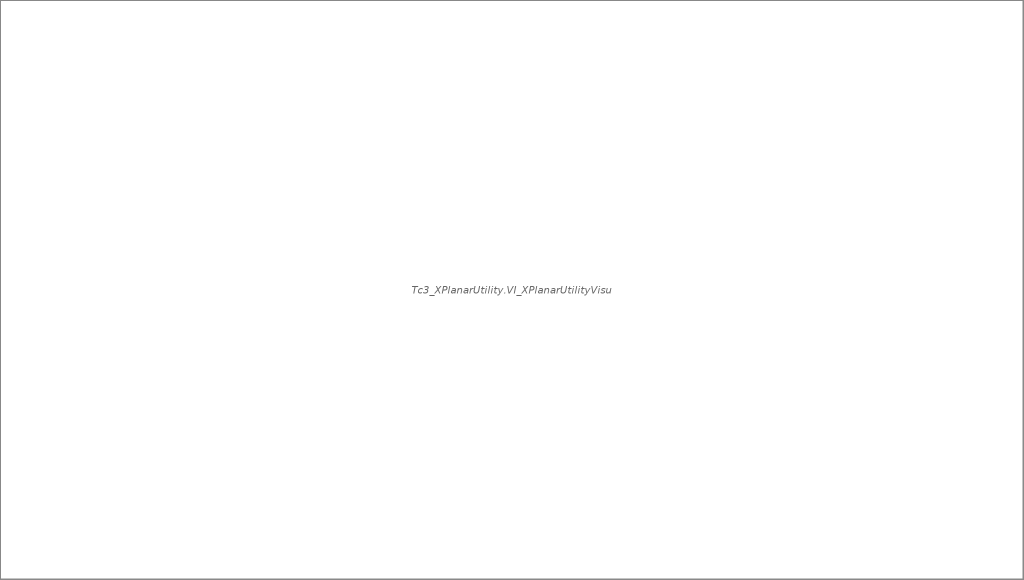
VISUALIZATION VI_Tc3_XPlanarUtility  // 1024x580
    Frame (0,0 1024x580)
        shows Tc3_XPlanarUtility.VI_XPlanarUtilityVisu()
END_VISUALIZATION

// ---- VISU/Visualization.TcVIS
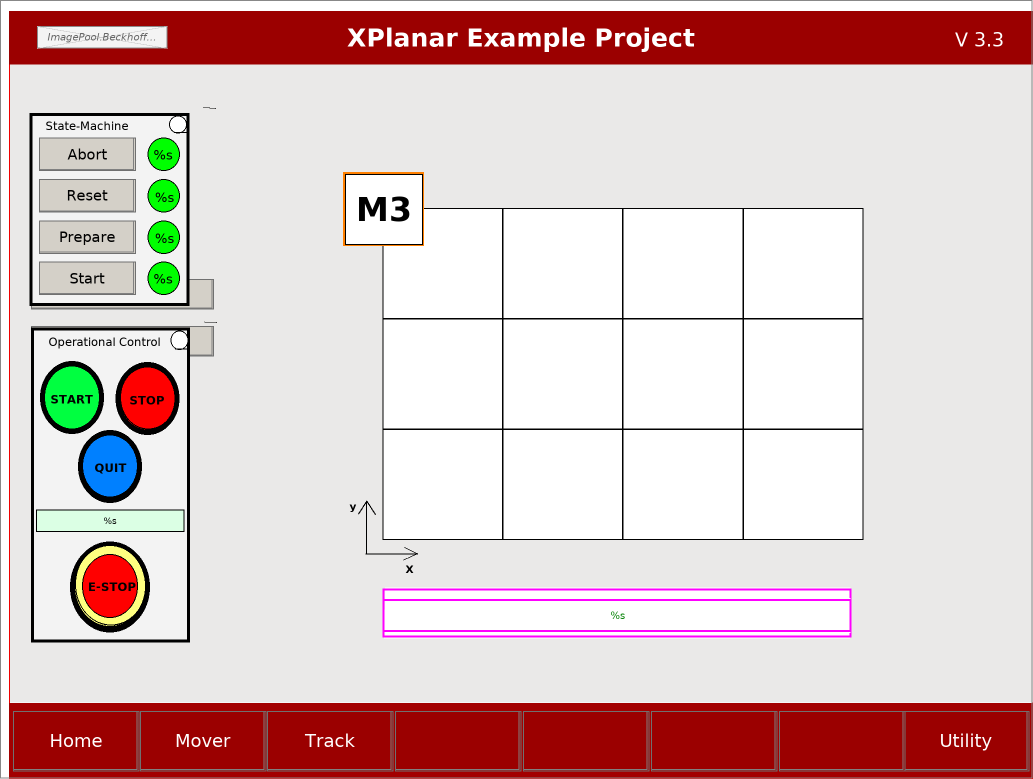
VISUALIZATION Visualization  // 1033x779
    Rectangle (9,11 1024x768)
    Frame (10,57 1023x645)
        shows VI_MainSide()
        shows Tc3_XPlanarStandard.VI_MoverLogOverview()
        shows Tc3_XPlanarStandard.VI_TrackLogOverview()
        shows VI_EtherCatDiag()
        shows VI_MoverDiag()
        shows VI_MoverTuning()
        shows VI_Tc3_XPlanarUtility()
        p1165984742: GVL_XtsVisu.pGroupRef[1]^.NcToPlc.Common.GroupStatus
        p547225198: GVL_XtsVisu.pGroupRef[1]
    Rectangle (9,703 1024x75)
    Button (13,711 126x60), "Home"
        OnMouseDown: FrameSelectionChange Selection=SelectedFrame=87eec691-4479-469a-bdd2-91ec7a1bb6bd, GlobSel=AssignType=Directly, SelType=Locally
    Button (140,711 126x60), "Mover"
        OnMouseUp: FrameSelectionChange Selection=SelectedFrame=87eec691-4479-469a-bdd2-91ec7a1bb6bd, Selection=1, GlobSel=AssignType=Directly, SelType=Locally
    Button (903,711 126x60), "Utility"
        OnMouseClick: change screen: UtilityPage
        OnMouseUp: change screen: UtilityPage
    Button (395,711 126x60)
    Button (523,711 126x60)
    Button (651,711 126x60)
    Button (779,711 126x60)
    Button (267,711 126x60), "Track"
        OnMouseUp: FrameSelectionChange Selection=SelectedFrame=87eec691-4479-469a-bdd2-91ec7a1bb6bd, Selection=2, GlobSel=AssignType=Expression, SelType=Locally
    Group (9,11 1024x53)
        Image (18,12 130x22), image: ImagePool.Beckhoff_white
        Image (18,11 130x22), image: ImagePool.Beckhoff_white
        Rectangle (0,0 1024x53), "XPlanar Example Project"
        Image (28,15 130x22), image: ImagePool.Beckhoff_white
        Rectangle (928,15 85x28), "V 3.3"
END_VISUALIZATION
